FUNCTION f_MoverIdDetectionModeToString : string(20)
VAR_INPUT
  nDetectionMode    : UINT;
END_VAR
VAR
END_VAR


CASE nDetectionMode
OF
  0:
    f_MoverIdDetectionModeToString  := 'Standard';
  1:
    f_MoverIdDetectionModeToString  := 'Mover 1';
  2:
    f_MoverIdDetectionModeToString  := 'Multiple Mover 1';
ELSE
    f_MoverIdDetectionModeToString  := 'UNKNOWN Mode';
END_CASE

END_FUNCTION

(* stored: Version 1.1.0.1, ProductVersion 3.1.4024.12
   POU f_MoverIdDetectionModeToString: Id {7e1d0e8e-62c8-48d1-9841-1d02395e8d1a}, SpecialFunc None *)
